% RSLogix 500 project 10.3.RSS, saved by version 8.30.00.16 %
PROJECT "10.3"    % processor: Bul.1763 MicroLogix 1100 Series B %

PROGRAM FILES
  LAD 2   4 rungs

DATA FILES
  O0 OUTPUT  4 elements
  I1 INPUT  6 elements
  S2 STATUS  66 elements
  B3 BINARY  1 elements
  T4 TIMER  1 elements
  C5 COUNTER  1 elements
  R6 CONTROL  1 elements
  N7 INTEGER  7 elements
  F8 FLOAT  1 elements

LADDER 2
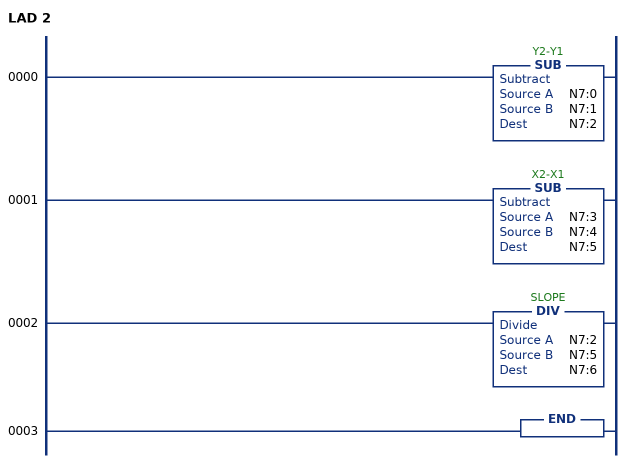
% Rung: 0 %
SOR SUB N7:0 N7:1 N7:2 EOR
%   N7:1  "Y1" %
%   N7:2  "Y2-Y1" %
% Rung: 1 %
SOR SUB N7:3 N7:4 N7:5 EOR
%   N7:5  "X2-X1" %
% Rung: 2 %
SOR DIV N7:2 N7:5 N7:6 EOR
%   N7:2  "Y2-Y1" %
%   N7:5  "X2-X1" %
%   N7:6  "SLOPE" %
% Rung: 3 %
SOR END EOR

DATA TABLE (non-zero values as saved)
DATA N7
% N7:0 % 15 10 0 10 5 0 0
